(* Logix 5000 project; controller prueba_de_git vendor 1 type 14 code 3 rev 13.1; software revision 13.04 *)

TASK MainTask (continuous, watchdog 500 ms) : MainProgram

MODULES
   Local : vendor 1 type 14 code 3 (ICP 0, rev 13.1)
END_MODULES

VAR_GLOBAL   (* controller tags *)
   B3 : DINT;
END_VAR

PROGRAM MainProgram   (* routine attr 65 MainRoutine *)

ROUTINE MainRoutine   (* ladder *)
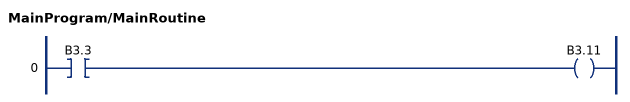
   0: XIC(B3.3)OTE(B3.11);
END_ROUTINE
END_PROGRAM
